// Mitsubishi GX Works2 project: 8182개 초기화   PLC: Q02/Q02H

PROGRAM MAIN
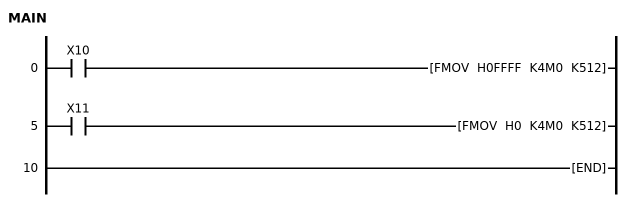
0     LD      X10
      FMOV    H0FFFF K4M0 K512
5     LD      X11
      FMOV    H0 K4M0 K512
10    END
END_PROGRAM
